(* IEC 61131-3 sources: ICSQuartz/benchmarks/scan_cycle_aircraft_oobr/src, 1 file *)

(* ---- program.st ---- *)
VAR_GLOBAL CONSTANT
    SS_INITIALIZE: SINT := 0;
    SS_STEP: SINT := 1;
    SS_FIN: SINT := 2;
END_VAR

PROGRAM PLC_PRG
VAR_INPUT
	In: ARRAY[0..7] OF LREAL := [3.0, 2.0, 3.0, 4.0, 1.0, 0.0, -1.0, 2.5];
    ssMethodType: SINT := SS_INITIALIZE;
END_VAR
VAR
	Out: ARRAY[0..1] OF LREAL;
    Code: Code;
END_VAR

// Harness simulation
Code(In, ssMethodType);

END_PROGRAM

FUNCTION_BLOCK Code
VAR_IN_OUT
    InRecv: ARRAY[0..7] OF LREAL;
    ssMethodType: SINT;
END_VAR
VAR
	offset: DWORD;
    CycleCount: INT;
	wGust: LREAL;
    qGust: LREAL;
    iter: INT;
	In: ARRAY[0..64] OF LREAL;
END_VAR
VAR_OUTPUT
    Out: ARRAY[0..1] OF LREAL;
END_VAR

// Complex branching logic
CASE ssMethodType OF

    SS_INITIALIZE:
        // Initialize memory
        FOR iter := 0 TO 64 DO
            In[iter] := 0.0;
        END_FOR;
        ssMethodType := SS_STEP;

    SS_STEP:

        // Copy Inputs
        CycleCount := CycleCount + 1;
        MemCpy(ADR(In), ADR(InRecv), offset);
        wGust := In[0];
        qGust := In[1];

        // Trigger potential memory error (oob read/write)
        // printf('cycle count: %d$N', CycleCount);
        // printf('offset: %d$N', offset);
        IF InRecv[0] > 1.1 AND InRecv[0] < 1.5 AND InRecv[1] > 2 AND InRecv[1] < 2.14 AND InRecv[2] > 5 AND InRecv[2] < 6.5 THEN
            IF CycleCount MOD 2 = 0 THEN
                offset := offset + 10;
            END_IF
        END_IF
        // IF In[CycleCount MOD 64] > 10 THEN
        //     In[CycleCount MOD 64 + 1] := In[CycleCount MOD 64 + 1] * 1.5;
        // ELSE
        //     In[CycleCount MOD 64 + 2] := In[CycleCount MOD 64 + 2] / 0.5;
        // END_IF;

        // More branching
        IF InRecv[2] < 3.5 AND InRecv[2] > 3.01 THEN
            In[3] := In[3] - 0.7;
            IF CycleCount MOD 2 = 0 THEN
                ssMethodType := SS_FIN;
            END_IF
        ELSE
            In[4] := In[4] + 0.8;
            IF In[4] > 1.0 AND IN[4] < 10.0 THEN
                In[5] := In[5] - 0.5;
                // ssMethodType := SS_FIN;
            ELSE
                In[5] := In[5] + 0.5;
                // ssMethodType := SS_INITIALIZE;
            END_IF;
        END_IF;

        // Additional logic for memory error
        IF In[5] < -1.0 THEN
            In[6] := In[6] * 2.0;
            // ssMethodType := SS_FIN;
        ELSE
            In[7] := In[7] / 2.0;
            // offset := offset - 1;
        END_IF;

        // Outputs for Atomic SubSystem: '<Root>/Code 2'
        Out[0] := -0.6385 * wGust;
        Out[1] := (-0.00592 * wGust) + (-0.6571 * qGust);

    SS_FIN:
        // No action
END_CASE;

END_FUNCTION_BLOCK
